# EPICS substitutions: apps/richsimApp/Db/TEMPRICH.substitutions
file "db/richtemp_sim.db" {
        pattern { Cr,    CrName,         CrType, Sl,     Ch,    Sys,     Det,    Element,        	CScode }
                {"17",  "TEMPRICH",	"4527", "08",   "00",   "TEMP",   "RICH", "SEC1_ROW1_PANEL1",	"#C2065"}
                {"17",  "TEMPRICH",	"4527", "08",   "01",   "TEMP",   "RICH", "SEC1_ROW1_PANEL2",	"#C2065"}
                {"17",  "TEMPRICH",	"4527", "08",   "02",   "TEMP",   "RICH", "SEC1_ROW1_PANEL3",	"#C2065"}
                {"17",  "TEMPRICH",	"4527", "08",   "03",   "TEMP",   "RICH", "SEC1_ROW1_PANEL4",	"#C2065"}
                {"17",  "TEMPRICH",	"4527", "08",   "04",   "TEMP",   "RICH", "SEC1_ROW1_PANEL5",	"#C2065"}
                {"17",  "TEMPRICH",	"4527", "08",   "05",   "TEMP",   "RICH", "SEC1_ROW1_PANEL6",	"#C2065"}
                {"17",  "TEMPRICH",	"4527", "08",   "06",   "TEMP",   "RICH", "SEC1_ROW1_PANEL7",	"#C2065"}
                {"17",  "TEMPRICH",	"4527", "08",   "07",   "TEMP",   "RICH", "SEC1_ROW1_PANEL8",	"#C2065"}
                {"17",  "TEMPRICH",	"4527", "08",   "08",   "TEMP",   "RICH", "SEC1_ROW1_PANEL9",	"#C2065"}
                {"17",  "TEMPRICH",	"4527", "08",   "09",   "TEMP",   "RICH", "SEC1_ROW1_PANEL10",	"#C2065"}
                {"17",  "TEMPRICH",	"4527", "08",   "10",   "TEMP",   "RICH", "SEC1_ROW2_PANEL1",	"#C2065"}
                {"17",  "TEMPRICH",	"4527", "08",   "11",   "TEMP",   "RICH", "SEC1_ROW2_PANEL2",	"#C2065"}
                {"17",  "TEMPRICH",	"4527", "08",   "12",   "TEMP",   "RICH", "SEC1_ROW2_PANEL3",	"#C2065"}
                {"17",  "TEMPRICH",	"4527", "08",   "13",   "TEMP",   "RICH", "SEC1_ROW2_PANEL4",	"#C2065"}
                {"17",  "TEMPRICH",	"4527", "08",   "14",   "TEMP",   "RICH", "SEC1_ROW2_PANEL5",	"#C2065"}
                {"17",  "TEMPRICH",	"4527", "08",   "15",   "TEMP",   "RICH", "SEC1_ROW2_PANEL6",	"#C2065"}
                {"17",  "TEMPRICH",	"4527", "08",   "16",   "TEMP",   "RICH", "SEC1_ROW2_PANEL7",	"#C2065"}
                {"17",  "TEMPRICH",	"4527", "08",   "17",   "TEMP",   "RICH", "SEC1_ROW2_PANEL8",	"#C2065"}
                {"17",  "TEMPRICH",	"4527", "08",   "18",   "TEMP",   "RICH", "SEC1_ROW2_PANEL9",	"#C2065"}
                {"17",  "TEMPRICH",	"4527", "08",   "19",   "TEMP",   "RICH", "SEC1_ROW3_PANEL1",	"#C2065"}
                {"17",  "TEMPRICH",	"4527", "08",   "20",   "TEMP",   "RICH", "SEC1_ROW3_PANEL2",	"#C2065"}
                {"17",  "TEMPRICH",	"4527", "08",   "21",   "TEMP",   "RICH", "SEC1_ROW3_PANEL3",	"#C2065"}
                {"17",  "TEMPRICH",	"4527", "08",   "22",   "TEMP",   "RICH", "SEC1_ROW3_PANEL4",	"#C2065"}
                {"17",  "TEMPRICH",	"4527", "08",   "23",   "TEMP",   "RICH", "SEC1_ROW3_PANEL5",	"#C2065"}
                {"17",  "TEMPRICH",	"4527", "08",   "24",   "TEMP",   "RICH", "SEC1_ROW3_PANEL6",	"#C2321"}
                {"17",  "TEMPRICH",	"4527", "08",   "25",   "TEMP",   "RICH", "SEC1_ROW3_PANEL7",	"#C2321"}
                {"17",  "TEMPRICH",	"4527", "08",   "26",   "TEMP",   "RICH", "SEC1_ROW3_PANEL8",	"#C2321"}
                {"17",  "TEMPRICH",	"4527", "08",   "27",   "TEMP",   "RICH", "SEC1_ROW3_PANEL9",	"#C2321"}
                {"17",  "TEMPRICH",	"4527", "08",   "28",   "TEMP",   "RICH", "SEC1_ROW4_PANEL1",	"#C2321"}
                {"17",  "TEMPRICH",	"4527", "08",   "29",   "TEMP",   "RICH", "SEC1_ROW4_PANEL2",	"#C2321"}
                {"17",  "TEMPRICH",	"4527", "08",   "30",   "TEMP",   "RICH", "SEC1_ROW4_PANEL3",	"#C2321"}
                {"17",  "TEMPRICH",	"4527", "08",   "31",   "TEMP",   "RICH", "SEC1_ROW4_PANEL4",	"#C2321"}
                {"17",  "TEMPRICH",	"4527", "08",   "32",   "TEMP",   "RICH", "SEC1_ROW4_PANEL5",	"#C2321"}
                {"17",  "TEMPRICH",	"4527", "08",   "33",   "TEMP",   "RICH", "SEC1_ROW4_PANEL6",	"#C2321"}
                {"17",  "TEMPRICH",	"4527", "08",   "34",   "TEMP",   "RICH", "SEC1_ROW4_PANEL7",	"#C2321"}
                {"17",  "TEMPRICH",	"4527", "08",   "35",   "TEMP",   "RICH", "SEC1_ROW4_PANEL8",	"#C2321"}
                {"17",  "TEMPRICH",	"4527", "08",   "36",   "TEMP",   "RICH", "SEC1_ROW4_PANEL9",	"#C2321"}
                {"17",  "TEMPRICH",	"4527", "08",   "37",   "TEMP",   "RICH", "SEC1_ROW5_PANEL1",	"#C2321"}
                {"17",  "TEMPRICH",	"4527", "08",   "38",   "TEMP",   "RICH", "SEC1_ROW5_PANEL2",	"#C2321"}
                {"17",  "TEMPRICH",	"4527", "08",   "39",   "TEMP",   "RICH", "SEC1_ROW5_PANEL3",	"#C2321"}
                {"17",  "TEMPRICH",	"4527", "08",   "40",   "TEMP",   "RICH", "SEC1_ROW5_PANEL4",	"#C2321"}
                {"17",  "TEMPRICH",	"4527", "08",   "41",   "TEMP",   "RICH", "SEC1_ROW5_PANEL5",	"#C2321"}
                {"17",  "TEMPRICH",	"4527", "08",   "42",   "TEMP",   "RICH", "SEC1_ROW5_PANEL6",	"#C2321"}
                {"17",  "TEMPRICH",	"4527", "08",   "43",   "TEMP",   "RICH", "SEC1_ROW5_PANEL7",	"#C2321"}
                {"17",  "TEMPRICH",	"4527", "08",   "44",   "TEMP",   "RICH", "SEC1_ROW5_PANEL8",	"#C2321"}
                {"17",  "TEMPRICH",	"4527", "08",   "46",   "TEMP",   "RICH", "SEC1_ROW6_PANEL1",	"#C2321"}
		{"17",  "TEMPRICH",     "4527", "08",   "47",   "TEMP",   "RICH", "SEC1_ROW6_PANEL2",   "#C2321"}
		{"17",  "TEMPRICH",     "4527", "08",   "48",   "TEMP",   "RICH", "SEC1_ROW6_PANEL3",   "#C2321"}
		{"17",  "TEMPRICH",     "4527", "08",   "49",   "TEMP",   "RICH", "SEC1_ROW6_PANEL4",   "#C2321"}
		{"17",  "TEMPRICH",     "4527", "08",   "50",   "TEMP",   "RICH", "SEC1_ROW6_PANEL5",   "#C2321"}
		{"17",  "TEMPRICH",     "4527", "08",   "51",   "TEMP",   "RICH", "SEC1_ROW6_PANEL6",   "#C2321"}
		{"17",  "TEMPRICH",     "4527", "08",   "52",   "TEMP",   "RICH", "SEC1_ROW6_PANEL7",   "#C2321"}
		{"17",  "TEMPRICH",     "4527", "08",   "53",   "TEMP",   "RICH", "SEC1_ROW6_PANEL8",   "#C2321"}
		{"17",  "TEMPRICH",     "4527", "08",   "54",   "TEMP",   "RICH", "SEC1_ROW7_PANEL1",   "#C2321"}
		{"17",  "TEMPRICH",     "4527", "08",   "55",   "TEMP",   "RICH", "SEC1_ROW7_PANEL2",   "#C2321"}
		{"17",  "TEMPRICH",     "4527", "08",   "56",   "TEMP",   "RICH", "SEC1_ROW7_PANEL3",   "#C2321"}
		{"17",  "TEMPRICH",     "4527", "08",   "57",   "TEMP",   "RICH", "SEC1_ROW7_PANEL4",   "#C2321"}
		{"17",  "TEMPRICH",     "4527", "08",   "58",   "TEMP",   "RICH", "SEC1_ROW7_PANEL5",   "#C2321"}
		{"17",  "TEMPRICH",     "4527", "08",   "59",   "TEMP",   "RICH", "SEC1_ROW7_PANEL6",   "#C2321"}
		{"17",  "TEMPRICH",     "4527", "08",   "60",   "TEMP",   "RICH", "SEC1_ROW7_PANEL7",   "#C2321"}
                {"17",  "TEMPRICH",     "4527", "08",   "61",   "TEMP",   "RICH", "SEC1_ROW7_PANEL8",   "#C2321"}
                {"17",  "TEMPRICH",     "4527", "08",   "62",   "TEMP",   "RICH", "SEC1_ROW8_PANEL1",   "#C2321"}
                {"17",  "TEMPRICH",     "4527", "08",   "63",   "TEMP",   "RICH", "SEC1_ROW8_PANEL2",   "#C2321"}
                {"17",  "TEMPRICH",     "4527", "08",   "64",   "TEMP",   "RICH", "SEC1_ROW8_PANEL3",   "#C2321"}
                {"17",  "TEMPRICH",     "4527", "08",   "65",   "TEMP",   "RICH", "SEC1_ROW8_PANEL4",   "#C2321"}
                {"17",  "TEMPRICH",     "4527", "08",   "66",   "TEMP",   "RICH", "SEC1_ROW8_PANEL5",   "#C2321"}
                {"17",  "TEMPRICH",     "4527", "08",   "67",   "TEMP",   "RICH", "SEC1_ROW8_PANEL6",   "#C2321"}
                {"17",  "TEMPRICH",     "4527", "08",   "68",   "TEMP",   "RICH", "SEC1_ROW8_PANEL7",   "#C2321"}
                {"17",  "TEMPRICH",     "4527", "08",   "69",   "TEMP",   "RICH", "SEC1_ROW9_PANEL1",   "#C2321"}
                {"17",  "TEMPRICH",     "4527", "08",   "70",   "TEMP",   "RICH", "SEC1_ROW9_PANEL2",   "#C2321"}
                {"17",  "TEMPRICH",     "4527", "08",   "71",   "TEMP",   "RICH", "SEC1_ROW9_PANEL3",   "#C2321"}
                {"17",  "TEMPRICH",     "4527", "08",   "72",   "TEMP",   "RICH", "SEC1_ROW9_PANEL4",   "#C2321"}
		{"17",  "TEMPRICH",     "4527", "08",   "73",   "TEMP",   "RICH", "SEC1_ROW9_PANEL5",   "#C2321"}
                {"17",  "TEMPRICH",     "4527", "08",   "74",   "TEMP",   "RICH", "SEC1_ROW9_PANEL6",   "#C2321"}
		{"17",  "TEMPRICH",     "4527", "08",   "75",   "TEMP",   "RICH", "SEC1_ROW9_PANEL7",   "#C2321"}
                {"17",  "TEMPRICH",     "4527", "08",   "76",   "TEMP",   "RICH", "SEC1_ROW10_PANEL1",  "#C2321"}
                {"17",  "TEMPRICH",     "4527", "08",   "77",   "TEMP",   "RICH", "SEC1_ROW10_PANEL2",  "#C2321"}
                {"17",  "TEMPRICH",     "4527", "08",   "78",   "TEMP",   "RICH", "SEC1_ROW10_PANEL3",  "#C2321"}
                {"17",  "TEMPRICH",     "4527", "08",   "79",   "TEMP",   "RICH", "SEC1_ROW10_PANEL4",  "#C2321"}
                {"17",  "TEMPRICH",     "4527", "08",   "80",   "TEMP",   "RICH", "SEC1_ROW10_PANEL5",  "#C2321"}
                {"17",  "TEMPRICH",     "4527", "08",   "81",   "TEMP",   "RICH", "SEC1_ROW10_PANEL6",  "#C2321"}
                {"17",  "TEMPRICH",     "4527", "08",   "82",   "TEMP",   "RICH", "SEC1_ROW10_PANEL7",  "#C2321"}
                {"17",  "TEMPRICH",     "4527", "08",   "83",   "TEMP",   "RICH", "SEC1_ROW11_PANEL1",  "#C2321"}
                {"17",  "TEMPRICH",     "4527", "08",   "84",   "TEMP",   "RICH", "SEC1_ROW11_PANEL2",  "#C2321"}
                {"17",  "TEMPRICH",     "4527", "08",   "85",   "TEMP",   "RICH", "SEC1_ROW11_PANEL3",  "#C2321"}
                {"17",  "TEMPRICH",     "4527", "08",   "86",   "TEMP",   "RICH", "SEC1_ROW11_PANEL4",  "#C2321"}
                {"17",  "TEMPRICH",     "4527", "08",   "87",   "TEMP",   "RICH", "SEC1_ROW11_PANEL5",  "#C2321"}
                {"17",  "TEMPRICH",     "4527", "08",   "88",   "TEMP",   "RICH", "SEC1_ROW11_PANEL6",  "#C2321"}
		{"17",  "TEMPRICH",     "4527", "08",   "89",   "TEMP",   "RICH", "SEC1_ROW12_PANEL1",  "#C2321"}
                {"17",  "TEMPRICH",     "4527", "08",   "90",   "TEMP",   "RICH", "SEC1_ROW12_PANEL2",  "#C2321"}
                {"17",  "TEMPRICH",     "4527", "08",   "91",   "TEMP",   "RICH", "SEC1_ROW12_PANEL3",  "#C2321"}
                {"17",  "TEMPRICH",     "4527", "08",   "92",   "TEMP",   "RICH", "SEC1_ROW12_PANEL4",  "#C2321"}
                {"17",  "TEMPRICH",     "4527", "08",   "93",   "TEMP",   "RICH", "SEC1_ROW12_PANEL5",  "#C2321"}
                {"17",  "TEMPRICH",     "4527", "08",   "94",   "TEMP",   "RICH", "SEC1_ROW12_PANEL6",  "#C2321"}
                {"17",  "TEMPRICH",     "4527", "08",   "95",   "TEMP",   "RICH", "SEC1_ROW13_PANEL1",  "#C2321"}
                {"17",  "TEMPRICH",     "4527", "08",   "96",   "TEMP",   "RICH", "SEC1_ROW13_PANEL2",  "#C2321"}
                {"17",  "TEMPRICH",     "4527", "08",   "97",   "TEMP",   "RICH", "SEC1_ROW13_PANEL3",  "#C2321"}
                {"17",  "TEMPRICH",     "4527", "08",   "98",   "TEMP",   "RICH", "SEC1_ROW13_PANEL4",  "#C2321"}
                {"17",  "TEMPRICH",     "4527", "08",   "99",   "TEMP",   "RICH", "SEC1_ROW13_PANEL5",  "#C2321"}
                {"17",  "TEMPRICH",     "4527", "08",   "100",   "TEMP",   "RICH", "SEC1_ROW13_PANEL6", "#C2321"}
                {"17",  "TEMPRICH",     "4527", "08",   "101",   "TEMP",   "RICH", "SEC1_ROW14_PANEL1", "#C2321"}
		{"17",  "TEMPRICH",	"4527", "08",   "102",   "TEMP",   "RICH", "SEC1_ROW14_PANEL2",	"#C2321"}
		{"17",  "TEMPRICH",	"4527", "08",   "103",   "TEMP",   "RICH", "SEC1_ROW14_PANEL3",	"#C2321"}
		{"17",  "TEMPRICH",	"4527", "08",   "104",   "TEMP",   "RICH", "SEC1_ROW14_PANEL4",	"#C2321"}
		{"17",  "TEMPRICH",	"4527", "08",   "105",   "TEMP",   "RICH", "SEC1_ROW14_PANEL5",	"#C2321"}
		{"17",  "TEMPRICH",	"4527", "08",   "106",   "TEMP",   "RICH", "SEC1_ROW15_PANEL1",	"#C2321"}
		{"17",  "TEMPRICH",	"4527", "08",   "107",   "TEMP",   "RICH", "SEC1_ROW15_PANEL2",	"#C2321"}
                {"17",  "TEMPRICH",	"4527", "08",   "108",   "TEMP",   "RICH", "SEC1_ROW15_PANEL3",	"#C2321"}
                {"17",  "TEMPRICH",	"4527", "08",   "109",   "TEMP",   "RICH", "SEC1_ROW15_PANEL4",	"#C2321"}
                {"17",  "TEMPRICH",	"4527", "08",   "110",   "TEMP",   "RICH", "SEC1_ROW15_PANEL5",	"#C2321"}
                {"17",  "TEMPRICH",	"4527", "08",   "111",   "TEMP",   "RICH", "SEC1_ROW16_PANEL1",	"#C2321"}
                {"17",  "TEMPRICH",	"4527", "08",   "112",   "TEMP",   "RICH", "SEC1_ROW16_PANEL2",	"#C2321"}
		{"17",  "TEMPRICH",	"4527", "08",   "113",   "TEMP",   "RICH", "SEC1_ROW16_PANEL3",	"#C2321"}
                {"17",  "TEMPRICH",	"4527", "08",   "114",   "TEMP",   "RICH", "SEC1_ROW16_PANEL4",	"#C2321"}
                {"17",  "TEMPRICH",	"4527", "08",   "115",   "TEMP",   "RICH", "SEC1_ROW16_PANEL5",	"#C2321"}
                {"17",  "TEMPRICH",	"4527", "08",   "116",   "TEMP",   "RICH", "SEC1_ROW17_PANEL1",	"#C2321"}
                {"17",  "TEMPRICH",	"4527", "08",   "117",   "TEMP",   "RICH", "SEC1_ROW17_PANEL2",	"#C2321"}
                {"17",  "TEMPRICH",	"4527", "08",   "118",   "TEMP",   "RICH", "SEC1_ROW17_PANEL3",	"#C2321"}
		{"17",  "TEMPRICH",	"4527", "08",   "119",   "TEMP",   "RICH", "SEC1_ROW17_PANEL4",	"#C2321"}
                {"17",  "TEMPRICH",	"4527", "08",   "120",   "TEMP",   "RICH", "SEC1_ROW18_PANEL1",	"#C2321"}
                {"17",  "TEMPRICH",	"4527", "08",   "121",   "TEMP",   "RICH", "SEC1_ROW18_PANEL2",	"#C2321"}
                {"17",  "TEMPRICH",	"4527", "08",   "122",   "TEMP",   "RICH", "SEC1_ROW18_PANEL3",	"#C2321"}
                {"17",  "TEMPRICH",	"4527", "08",   "123",   "TEMP",   "RICH", "SEC1_ROW18_PANEL4",	"#C2321"}
                {"17",  "TEMPRICH",	"4527", "08",   "124",   "TEMP",   "RICH", "SEC1_ROW19_PANEL1",	"#C2321"}
		{"17",  "TEMPRICH",	"4527", "08",   "125",   "TEMP",   "RICH", "SEC1_ROW19_PANEL2",	"#C2321"}
                {"17",  "TEMPRICH",	"4527", "08",   "126",   "TEMP",   "RICH", "SEC1_ROW19_PANEL3",	"#C2321"}
                {"17",  "TEMPRICH",	"4527", "08",   "127",   "TEMP",   "RICH", "SEC1_ROW19_PANEL4",	"#C2321"}
                {"17",  "TEMPRICH",	"4527", "08",   "128",   "TEMP",   "RICH", "SEC1_ROW20_PANEL1",	"#C2321"}
                {"17",  "TEMPRICH",	"4527", "08",   "129",   "TEMP",   "RICH", "SEC1_ROW20_PANEL2",	"#C2321"}
                {"17",  "TEMPRICH",	"4527", "08",   "130",   "TEMP",   "RICH", "SEC1_ROW20_PANEL3",	"#C2321"}
		{"17",  "TEMPRICH",	"4527", "08",   "131",   "TEMP",   "RICH", "SEC1_ROW21_PANEL1",	"#C2321"}
                {"17",  "TEMPRICH",	"4527", "08",   "132",   "TEMP",   "RICH", "SEC1_ROW21_PANEL2",	"#C2321"}
                {"17",  "TEMPRICH",	"4527", "08",   "133",   "TEMP",   "RICH", "SEC1_ROW21_PANEL3",	"#C2321"}
                {"17",  "TEMPRICH",	"4527", "08",   "134",   "TEMP",   "RICH", "SEC1_ROW22_PANEL1",	"#C2321"}
                {"17",  "TEMPRICH",	"4527", "08",   "135",   "TEMP",   "RICH", "SEC1_ROW22_PANEL2",	"#C2321"}
                {"17",  "TEMPRICH",	"4527", "08",   "136",   "TEMP",   "RICH", "SEC1_ROW22_PANEL3",	"#C2321"}
		{"17",  "TEMPRICH",	"4527", "08",   "137",   "TEMP",   "RICH", "SEC1_ROW23_PANEL1",	"#C2321"}
                {"17",  "TEMPRICH",	"4527", "08",   "138",   "TEMP",   "RICH", "SEC1_ROW23_PANEL2",	"#C2321"}
}
